(* IEC 61131-3 sources: Industry-PLC-LLM/data/PLCBEAD_repo/PLCBEAD_PLCEmbed-main/PLC-BEAD/Source/GEB/LEAP_YEAR, 1 file *)

(* ---- LEAP_YEAR.ST ---- *)
FUNCTION LEAP_YEAR:BOOL

  VAR_INPUT
    YEAR  :	INT;
  END_VAR

  IF (YEAR  MOD INT#400) = INT#00 THEN
    LEAP_YEAR  := TRUE;
  ELSIF (YEAR  MOD INT#100) = INT#00 THEN
    LEAP_YEAR  := FALSE;
  ELSIF (YEAR  MOD INT#04) = INT#00 THEN
    LEAP_YEAR  := TRUE;
  ELSE
    LEAP_YEAR  := FALSE;
  END_IF;

END_FUNCTION

PROGRAM program0
	VAR
		YEAR  :	INT;
		OUT : BOOL;
	END_VAR

	OUT := LEAP_YEAR(YEAR);
END_PROGRAM
